Fanuc KAREL source: kb00008.KL

-- PROVISIONAL review KL for V770-1; original PC SHA256 5093d864e8940918da854d0fb91d447f7ac6768faab46637dddbb5a6d4d9d1ba
-- Incomplete behavior may be omitted. Consult companion uncertainty JSON. Do not deploy.
PROGRAM KB00008
%NOLOCKGROUP
VAR
  P1 : REAL
  RESULT : REAL
BEGIN
  -- UNRESOLVED_PC offsets 5-16; opcodes 2E,23
  -- UNRESOLVED_PC offsets 21-36; opcodes 27,22,76,23
  -- UNRESOLVED_PC offsets 41-45; opcodes 7F
END KB00008
